FUNCTION F_SAFETY_StatusFB_TO_TOF : ST_SAFETY_FBTOF
VAR_INPUT
	stFBStatus						: ST_SAFETY_FBStatus; 	(* Struktura ogolna *)
END_VAR

F_SAFETY_StatusFB_TO_TOF.uStatus.stStatusWords 		:= stFBStatus;									(* Przepisanie *)
F_SAFETY_StatusFB_TO_TOF.eState					 	:= stFBStatus.BState;							(* Ustawienie enum *)

END_FUNCTION

(* stored: Version 1.1.0.1, ProductVersion 3.1.4022.12
   POU F_SAFETY_StatusFB_TO_TOF: Id {884b2e69-8196-4dd6-9c06-72c4c25a3927}, SpecialFunc None *)
